// TwinCAT 3 PLC project
// project tree:
//   GVLs/ Plant.TcGVL
//   POUs/ MAIN.TcPOU

// ---- GVLs/Plant.TcGVL
VAR_GLOBAL
  MixerRenamed : FB_Device;
  FlowValue : REAL;
  NewlyAddedSensor : INT;
  ValveCommand : BOOL := FALSE;
END_VAR

// ---- POUs/MAIN.TcPOU
PROGRAM MAIN
VAR
  LocalPermit : BOOL;
END_VAR


Plant.MixerRenamed(Start := LocalPermit);
Plant.ValveCommand := LocalPermit;

END_PROGRAM
